(* CoDeSys 2.3.10.0 project: derevo.pr6 *)
(* Author: Yurko Shybaigolova *)
(* Libraries: STANDARD.LB6 5.6.98 13:03:02 *)

(* Global variable list: physical *)
(* @GLOBAL_VARIABLE_LIST := TwinCAT_Import *)
(* @PATH := '' *)
VAR_GLOBAL (* DO NOT CHANGE THIS SHEET MANUALLY! *)
	PlcInVar_0	AT %QB128:	USINT;
	PlcInVar_1	AT %QB129:	USINT;
	PlcInVar_2	AT %QB130:	USINT;
	PlcInVar_3	AT %QB131:	USINT;
	PlcInVar_4	AT %QB132:	USINT;
	PlcInVar_5	AT %QB133:	USINT;
	PlcInVar_6	AT %QB134:	USINT;
	PlcInVar_7	AT %QB135:	USINT;
	PlcInVar_8	AT %QB136:	USINT;
	PlcInVar_9	AT %QB137:	USINT;
	PlcInVar_10	AT %QB138:	USINT;
	PlcInVar_11	AT %QB139:	USINT;
	PlcInVar_12	AT %QB140:	USINT;
	PlcInVar_13	AT %QB141:	USINT;
	PlcInVar_14	AT %QB142:	USINT;
	PlcInVar_15	AT %QB143:	USINT;
	PlcOutVar_0	AT %IB128:	USINT;
	PlcOutVar_1	AT %IB129:	USINT;
	PlcOutVar_2	AT %IB130:	USINT;
	PlcOutVar_3	AT %IB131:	USINT;
	PlcOutVar_4	AT %IB132:	USINT;
	PlcOutVar_5	AT %IB133:	USINT;
	PlcOutVar_6	AT %IB134:	USINT;
	PlcOutVar_7	AT %IB135:	USINT;
	PlcOutVar_8	AT %IB136:	USINT;
	PlcOutVar_9	AT %IB137:	USINT;
	PlcOutVar_10	AT %IB138:	USINT;
	PlcOutVar_11	AT %IB139:	USINT;
	PlcOutVar_12	AT %IB140:	USINT;
	PlcOutVar_13	AT %IB141:	USINT;
	PlcOutVar_14	AT %IB142:	USINT;
	PlcOutVar_15	AT %IB143:	USINT;
	term1 AT%QB0:BYTE;
	term2 AT%QB1:BYTE;
	term3 AT%QB2:BYTE;
	term4 AT%QB3:BYTE;
	vidpochynok1	AT %QX0.0:	BOOL;
	vidpochynok2	AT %QX0.1:	BOOL;
	veranda 		AT %QX0.2:	BOOL;
	veranda_zovn	AT %QX0.3:	BOOL;
	vhid_zovn		AT %QX0.4:	BOOL;
	sauna			AT %QX0.5:	BOOL;
	vhid			AT %QX0.6:	BOOL;
	Term_2_KL2408_8_Output	AT %QX0.7:	BOOL;
	korydor			AT %QX1.0:	BOOL;
	sinna			AT %QX1.1:	BOOL;
	hamam			AT %QX1.2:	BOOL;
	kuhnya			AT %QX1.3:	BOOL;
	bassein1		AT %QX1.4:	BOOL;
	bassein2		AT %QX1.5:	BOOL;
	spalnya2	AT %QX1.6:	BOOL;
	terassa			AT %QX1.7:	BOOL;
	dush			AT %QX2.0:	BOOL;
	wc				AT %QX2.1:	BOOL;
	spalnya_verh	AT %QX2.2:	BOOL;
	spalnya1		AT %QX2.3:	BOOL;
	spalnya_su		AT %QX2.4:	BOOL;
	garderob		AT %QX2.5:	BOOL;
	Term_4_KL2408_7_Output	AT %QX2.6:	BOOL;
	Term_4_KL2408_8_Output	AT %QX2.7:	BOOL;

	sw_vidpochynok1			AT %IX0.0:	BOOL;
	sw_vidpochynok2			AT %IX0.1:	BOOL;
	sw_veranda1				AT %IX0.2:	BOOL;
	sw_veranda2				AT %IX0.3:	BOOL;
	sw_spalnya1				AT %IX0.4:	BOOL;
	sw_spalnya2				AT %IX0.5:	BOOL;
	sw_vhid1			AT %IX0.6:	BOOL;
	sw_vhid2			AT %IX0.7:	BOOL;
	sw_korydor1				AT %IX1.0:	BOOL;
	sw_korydor2				AT %IX1.1:	BOOL;
	sw_vidpochynok_skhody1	AT %IX1.2:	BOOL;
	sw_vidpochynok_skhody2	AT %IX1.3:	BOOL;
	sw_sauna1				AT %IX1.4:	BOOL;
	sw_sauna2				AT %IX1.5:	BOOL;
	sw_bassein1				AT %IX1.6:	BOOL;
	sw_bassein2				AT %IX1.7:	BOOL;
	sw_sauna_vhid2		AT %IX2.0:	BOOL;
	sw_sauna_vhid1		AT %IX2.1:	BOOL;
	sw_sinna1					AT %IX2.2:	BOOL;
	Term_7_KL1408_4_Input	AT %IX2.3:	BOOL;
	sw_spalnya_su				AT %IX2.4:	BOOL;
	sw_garderob				AT %IX2.5:	BOOL;
	sw_kuh1					AT %IX2.6:	BOOL;
	sw_kuh2					AT %IX2.7:	BOOL;
	Term_8_KL1408_1_Input	AT %IX3.0:	BOOL;
	sw_sinna						AT %IX3.1:	BOOL;
	sw_skhody_22					AT %IX3.2:	BOOL;
	sw_skhody_21					AT %IX3.3:	BOOL;
	sw_skhody_12					AT %IX3.4:	BOOL;
	sw_skhody_11					AT %IX3.5:	BOOL;
	sw_hamam					AT %IX3.6:	BOOL;
	sw_spalnya_verh			AT %IX3.7:	BOOL;
	Term_9_KL1408_1_Input	AT %IX4.0:	BOOL;
	Term_9_KL1408_2_Input	AT %IX4.1:	BOOL;
	Term_9_KL1408_3_Input	AT %IX4.2:	BOOL;
	Term_9_KL1408_4_Input	AT %IX4.3:	BOOL;
	Term_9_KL1408_5_Input	AT %IX4.4:	BOOL;
	Term_9_KL1408_6_Input	AT %IX4.5:	BOOL;
	Term_9_KL1408_7_Input	AT %IX4.6:	BOOL;
	Term_9_KL1408_8_Input	AT %IX4.7:	BOOL;
END_VAR

(* @OBJECT_END := TwinCAT_Import *)

VAR_GLOBAL
END_VAR

(* POU MAIN, ST *)
PROGRAM MAIN
VAR

	g_veranda				:	SWITCH;
	g_spalnya1				:	SWITCH;
	g_spalnya2				:	SWITCH;
	g_sauna_skhody1			:	SWITCH;
	g_sauna_skhody2			:	SWITCH;
	g_bassein_skhody1		:	SWITCH;
	g_bassein_skhody2		:	SWITCH;
	g_vidpochynok_skhody1	:	SWITCH;
	g_vidpochynok_skhody2	:	SWITCH;
	g_sauna_vhid1				:	SWITCH;
	g_sauna_vhid2				:	SWITCH;
	g_bassein1				:	SWITCH;
	g_bassein2				:	SWITCH;
	g_sauna_skhody2_1		:	SWITCH;
	g_sauna_skhody2_2		:	SWITCH;
	g_sinna					:	SWITCH;
	g_Term_7_KL1408_4_Input	:	SWITCH;
	g_spalnya_su				:	SWITCH;
	g_garderob				:	SWITCH;
	g_kuh1					:	SWITCH;
	g_kuh2					:	SWITCH;

	g_sinna1						:	SWITCH;
	g_skhody_22					:	SWITCH;
	g_skhody_21					:	SWITCH;
	g_skhody_12					:	SWITCH;
	g_skhody_11					:	SWITCH;
	g_hamam					:	SWITCH;

	delay: TIME;
	g_vidpochynok1: SWITCH;
	g_vidpochynok2: SWITCH;
	g_veranda1: SWITCH;
	g_zovn: SWITCH;
	g_korydor: SWITCH;
	g_bassein: SWITCH;
	g_terassa: SWITCH;
	g_vhid: SWITCH;
	g_dush: SWITCH;
	g_wc: SWITCH;
	g_sauna: SWITCH;
	g_vhid_zovn: SWITCH;

	F_polka:F_TRIG;
	R_polka: R_TRIG;

	g_spalnya_verh: SWITCH;
END_VAR
delay:=t#1s;
	g_vidpochynok1(IN:=sw_vidpochynok1  XOR sw_vidpochynok_skhody1 XOR sw_skhody_11, SWITCH_DELAY:=delay,Q_SHORT=>vidpochynok1);
	g_vidpochynok2(IN:=sw_vidpochynok2, SWITCH_DELAY:=delay,Q_SHORT=>vidpochynok2);
	g_kuh1	(IN:=sw_kuh1 , SWITCH_DELAY:=delay,Q_SHORT=>kuhnya);
	g_kuh2	(IN:=sw_kuh2, SWITCH_DELAY:=delay(*kuhnya_pidsvitka*));

	g_veranda(IN:=sw_veranda1, SWITCH_DELAY:=delay,Q_SHORT=>veranda);

	g_zovn(IN:=sw_veranda2, SWITCH_DELAY:=delay,Q_SHORT=>veranda_zovn);

	g_spalnya1	(MODE:='short&long',IN:=sw_spalnya1, SWITCH_DELAY:=delay,Q_SHORT=>spalnya1);

	g_spalnya_verh( IN:=sw_spalnya_verh, SWITCH_DELAY:=delay);


F_polka(CLK:=g_spalnya1.Q_LONG XOR g_spalnya_verh.Q_SHORT);
R_polka(CLK:=g_spalnya_verh.Q_SHORT XOR g_spalnya1.Q_LONG );
IF F_polka.Q OR R_polka.Q THEN spalnya_verh:= NOT spalnya_verh; END_IF

	g_spalnya2	(IN:=sw_spalnya2, SWITCH_DELAY:=delay,Q_SHORT=>spalnya2);

	g_bassein(IN:=sw_korydor1 XOR sw_skhody_12, SWITCH_DELAY:=delay,Q_SHORT=>bassein1);
bassein2:=bassein1;

	g_terassa(IN:=sw_vidpochynok_skhody2, SWITCH_DELAY:=delay,Q_SHORT=>terassa);

	g_korydor(IN:= sw_korydor2 XOR  sw_sauna_vhid2 , SWITCH_DELAY:=delay,Q_SHORT=>korydor);

	g_sauna	(IN:=sw_sauna2, SWITCH_DELAY:=delay,Q_SHORT=>sauna);

	g_wc(IN:=sw_bassein1 XOR sw_skhody_21, SWITCH_DELAY:=delay,Q_SHORT=>wc);

	g_dush (IN:=sw_bassein2 XOR sw_skhody_22, SWITCH_DELAY:=delay,Q_SHORT=>dush);

	g_spalnya_su(IN:=sw_spalnya_su, SWITCH_DELAY:=delay,Q_SHORT=>spalnya_su);

	g_garderob	(IN:=sw_garderob, SWITCH_DELAY:=delay,Q_SHORT=>garderob);

	g_sinna(IN:=sw_sinna, SWITCH_DELAY:=delay,Q_SHORT=>sinna);

	g_hamam(IN:=sw_hamam, SWITCH_DELAY:=delay,Q_SHORT=>hamam);

	g_vhid_zovn(IN:=sw_vhid1 ,SWITCH_DELAY:=delay,Q_SHORT=>vhid_zovn);
	g_vhid(IN:=sw_sauna_vhid1 XOR sw_vhid2, SWITCH_DELAY:=delay,Q_SHORT=>vhid);
END_PROGRAM

(* POU Vymykachi/SWITCH, ST *)
FUNCTION_BLOCK SWITCH
VAR_INPUT
	IN:BOOL;
	SWITCH_DELAY:TIME; (*різниця між коротким і довгим натисненням*)
	SHORT_OFF_DELAY, LONG_OFF_DELAY: TIME; (*час затримки вимкнення по короткому та довгому натисненню*)
	MODE:STRING; (*delayed, light, light&vent, short&long, delayed_short&long, *)
	NUMBER_OF_OUTS:INT;
END_VAR
VAR_OUTPUT
	Q_SHORT:BOOL:=FALSE;
	Q_SHORT_D: BOOL;(*вихід для вимкнення із затримкою, вмикається разом із виходом короткого натискання*)
	Q_LONG:BOOL:=FALSE;
	Q_LONG_D:BOOL; (*вихід для вимкнення із затримкою, вмикається разом із виходом довгого натискання*)
END_VAR
VAR
	STAN:BOOL:=FALSE;
	Q_S_fall:F_TRIG; (*ловить задній фронт вихода короткого натискання*)
	Q_L_fall:F_TRIG;(*ловить задній фронт вихода довгого натискання*)
	chas: TIME; (*час доки кнопка натиснена*)

	long: BOOL; (*стає тру, якщо було довге натиснення*)
	short: BOOL; (*стає тру, якщо було коротке натиснення*)
	timer, short_off_delay_timer, long_off_delay_timer: TON; (*таймери: час натискання, час переключення відкладеного виходу по довгому та короткому натисканнях*)
	up: BOOL; (*кнопка натиснена*)

	delay_l, delay_s:BOOL; (*запускати таймери відкладеного вимкнення*)

	turn_off_long: BOOL;
	start_l, start_s:BOOL;
END_VAR
short:=0;
long:=0;
timer(IN:=IN AND STAN, PT:=t#10s);
IF IN AND STAN THEN
	chas:=timer.ET;
	up:=1;
ELSE
up:=0;
END_IF;

IF NOT IN AND NOT STAN THEN
chas:=t#0ms;
END_IF;

IF STAN AND NOT IN THEN
	IF chas <SWITCH_DELAY THEN
		short:=1;
		Q_SHORT:= NOT Q_SHORT;
	END_IF;
	IF chas>=SWITCH_DELAY THEN
		Q_LONG:= NOT Q_LONG;
		long:=1;
	END_IF;
END_IF;

(*затримка вимикання*)
Q_L_fall(CLK:=Q_LONG);
Q_S_fall(CLK:=Q_SHORT);

IF Q_L_FALL.Q THEN
		start_l:=TRUE;
END_IF

IF Q_S_FALL.Q THEN
	start_s:=TRUE;
END_IF

IF MODE='light&vent' THEN
	IF start_s THEN start_l:=start_s; END_IF
END_IF

IF LONG_OFF_DELAY <> t#0ms THEN (*виконувати лише якщо в блок переданий параметр затримки на вимкнення*)

	IF Q_LONG THEN
		Q_LONG_D:=Q_LONG;
	END_IF

	long_off_delay_timer(IN:=start_l, PT:=LONG_OFF_DELAY);

	IF long_off_delay_timer.Q THEN
		Q_LONG_D:=FALSE;
		start_l:=FALSE;
	END_IF

ELSE
	Q_LONG_D:=Q_LONG;
END_IF

IF SHORT_OFF_DELAY <> t#0ms THEN (*виконувати лише якщо в блок переданий параметр затримки на вимкнення*)

	IF Q_SHORT THEN
		Q_SHORT_D:=Q_SHORT;
	END_IF

	short_off_delay_timer(IN:=start_s, PT:=SHORT_OFF_DELAY);

	IF short_off_delay_timer.Q THEN
		Q_SHORT_D:=FALSE;
		start_s:=FALSE;
	END_IF


ELSE
	Q_SHORT_D:=Q_SHORT;
END_IF

IF MODE='delayed' THEN
	Q_LONG:=Q_LONG_D;
	Q_SHORT:=Q_SHORT_D;
END_IF
(*працють лише короткі замикання*)
IF MODE='light' THEN
	Q_SHORT_D:=FALSE;
	Q_LONG:=Q_SHORT;
	Q_LONG_D:=FALSE;
END_IF
(*затримки не працюють*)
IF MODE='short&long' THEN
	Q_SHORT_D:=FALSE;
	Q_LONG_D:=FALSE;
END_IF
(*при вимкненні всього світла вимикати вентилятор і затримкою*)
IF MODE='light&vent' THEN
	IF NOT Q_SHORT AND Q_LONG THEN
		Q_LONG:=Q_LONG_D;
	END_IF
END_IF

STAN := IN;
END_FUNCTION_BLOCK
